TYPE ST_HMI_SolventAndTimeRow  :
STRUCT
	Parameter : STRING(16);
    Rinse1    : INT;
    Rinse2    : INT;
    Wash1     : INT;
    Wash2     : INT;
END_STRUCT
END_TYPE

(* stored: Version 1.1.0.1, ProductVersion 3.1.4024.12
   DUT ST_HMI_SolventAndTimeRow: Id {673cd567-fb0a-4c11-95ab-37a7dfad03b2} *)
